# B&R Automation Studio project ComauRacer3demo (part 3)

### Main.st - not listed in the package file held
```iecst
PROGRAM _INIT
	cmd.MpFileManagerUI_0.MpLink := ADR(gFileManagerUI);
	cmd.MpFileManagerUI_0.Enable := TRUE;

	cmd.MpFileManagerUI_0.UISetup := cmd.MpFileManagerUISetupType;
	cmd.MpFileManagerUI_0.UIConnect := ADR(cmd.MpFileManagerUIConnectType);

	(* define of device names *)
	cmd.MpFileManagerUIConnectType.DeviceList.DeviceNames[0] := 'CNC_PrgDir';
	cmd.MpFileManagerUIConnectType.DeviceList.DeviceNames[1] := 'UserPart';
	cmd.MpFileManagerUIConnectType.DeviceList.DeviceNames[2] := 'AUDIT';
	cmd.MpFileManagerUIConnectType.DeviceList.DeviceNames[3] := 'RECIPE'; //currently not implemented

	cmd.MpFileManagerUIConnectType.File.NewName := '';

	cmd.MpFileManagerUI_0();
END_PROGRAM

PROGRAM _CYCLIC
	tabInfo.NumberOfElements := 0;
	FOR iFile := 0 TO 49 BY 1 DO
		(* create arrays with file properties *)
		brsmemcpy(ADR(tabInfo.Name[iFile]), ADR(cmd.MpFileManagerUIConnectType.File.List.Items[iFile].Name), SIZEOF(tabInfo.Name[iFile]));
		brsmemcpy(ADR(tabInfo.Size[iFile]), ADR(cmd.MpFileManagerUIConnectType.File.List.Items[iFile].Size), SIZEOF(tabInfo.Size[iFile]));
		brsmemcpy(ADR(tabInfo.Type[iFile]), ADR(cmd.MpFileManagerUIConnectType.File.List.Items[iFile].ItemType), SIZEOF(tabInfo.Type[iFile]));
		brsmemcpy(ADR(tabInfo.LastModified[iFile]), ADR(cmd.MpFileManagerUIConnectType.File.List.Items[iFile].LastModified), SIZEOF(tabInfo.LastModified[iFile]));

		IF tabInfo.SelectedRow = iFile THEN
			cmd.MpFileManagerUIConnectType.File.List.Items[iFile].IsSelected := TRUE;
		END_IF

		(* numbers of elements in the table *)
		IF tabInfo.Type[iFile] <> mpFILE_ITEM_TYPE_NONE THEN
			tabInfo.NumberOfElements := tabInfo.NumberOfElements + 1;
		END_IF
	END_FOR

	(* dynamic change of the array size *)
	brsitoa(tabInfo.NumberOfElements, ADR(aux.NumberOfElementsStr));
	aux.TableConfigurationStr := '{"specRows": [ {"from":0, "to":';
	aux.One := ', "visible":true}, {"from":';
	aux.Two := ', "to":49, "visible":false}]}';
	brsstrcat(ADR(aux.TableConfigurationStr), ADR(aux.NumberOfElementsStr));
	brsstrcat(ADR(aux.TableConfigurationStr), ADR(aux.One));
	brsstrcat(ADR(aux.TableConfigurationStr), ADR(aux.NumberOfElementsStr));
	brsstrcat(ADR(aux.TableConfigurationStr), ADR(aux.Two));

	aux.NumberOfElementsMinus := tabInfo.NumberOfElements - 1;

	IF tabInfo.NumberOfElements >= 1 THEN
		aux.NewNamePlus := 0;
		aux.newNewName := '';
		aux.prevNewName := cmd.MpFileManagerUIConnectType.File.NewName;
		aux.newNewName := aux.prevNewName;
		FOR iFile := 0 TO aux.NumberOfElementsMinus BY 1 DO
			(* dynamic change of the existing name *)
			IF tabInfo.Name[iFile] = aux.newNewName THEN
				aux.newNewName := aux.prevNewName;
				aux.NewNamePlus := aux.NewNamePlus + 1;
				brsitoa(aux.NewNamePlus, ADR(aux.NewNamePlusStr));
				aux.NewNameTextOne := '(';
				aux.NewNameTextTwo := ')';
				brsstrcat(ADR(aux.newNewName), ADR(aux.NewNameTextOne));
				brsstrcat(ADR(aux.newNewName), ADR(aux.NewNamePlusStr));
				brsstrcat(ADR(aux.newNewName), ADR(aux.NewNameTextTwo));
				//iFile := 0;
			ELSE
				cmd.MpFileManagerUIConnectType.File.NewName := aux.newNewName;
			END_IF
		END_FOR
	END_IF

	(* search engine *)
	cmd.MpFileManagerUIConnectType.File.Filter := '*';
	IF aux.SearchNewName <> '' THEN
		brsstrcat(ADR(cmd.MpFileManagerUIConnectType.File.Filter), ADR(aux.SearchNewName));
		brsstrcat(ADR(cmd.MpFileManagerUIConnectType.File.Filter), ADR(aux.textStar));
		cmd.MpFileManagerUIConnectType.File.Refresh := TRUE;
	ELSE
		cmd.MpFileManagerUIConnectType.File.Filter := '*';
	END_IF

	//change sorting method
	CASE aux.btnSort OF
		0:
			cmd.MpFileManagerUIConnectType.File.SortOrder := mpFILE_SORT_BY_NAME_ASC;
			aux.btnSortStr := '$$IAT/Browser/SortByNameAsc';
		1:
			cmd.MpFileManagerUIConnectType.File.SortOrder := mpFILE_SORT_BY_NAME_DESC;
			aux.btnSortStr := '$$IAT/Browser/SortByNameDesc';
		2:
			cmd.MpFileManagerUIConnectType.File.SortOrder := mpFILE_SORT_BY_SIZE_ASC;
			aux.btnSortStr := '$$IAT/Browser/SortBySizeAsc';
		3:
			cmd.MpFileManagerUIConnectType.File.SortOrder := mpFILE_SORT_BY_SIZE_DES;
			aux.btnSortStr := '$$IAT/Browser/SortBySizeDesc';
		4:
			cmd.MpFileManagerUIConnectType.File.SortOrder := mpFILE_SORT_BY_MOD_TIME_ASC;
			aux.btnSortStr := '$$IAT/Browser/SortByLastModAsc';
		5:
			cmd.MpFileManagerUIConnectType.File.SortOrder := mpFILE_SORT_BY_MOD_TIME_DESC;
			aux.btnSortStr := '$$IAT/Browser/SortByLastModDesc';
		6:
			aux.btnSort := 0;
	END_CASE

	//variables used to load files
	aux.fileName := tabInfo.Name[tabInfo.SelectedRow];
	aux.NewNameTextOne := '/';
	aux.fullFilePath := '';
	aux.fullFilePathWithFileDevice := '/FileDevice:';
	IF brsstrcmp(ADR(aux.fullFilePath), ADR(cmd.MpFileManagerUIConnectType.File.PathInfo.CurrentDir)) = 0 THEN //theoritically it works without it, but adds two '//' when not in a subfolder
		brsstrcat(ADR(aux.fullFilePath), ADR(cmd.MpFileManagerUIConnectType.DeviceList.DeviceNames[cmd.MpFileManagerUIConnectType.DeviceList.SelectedIndex])); //device name
		brsstrcat(ADR(aux.fullFilePath), ADR(aux.NewNameTextOne)); // '/'
		brsstrcat(ADR(aux.fullFilePath), ADR(aux.fileName)); // file name, this gives full file path in subsystem.
	ELSE
		brsstrcat(ADR(aux.fullFilePath), ADR(cmd.MpFileManagerUIConnectType.DeviceList.DeviceNames[cmd.MpFileManagerUIConnectType.DeviceList.SelectedIndex])); //device name
		brsstrcat(ADR(aux.fullFilePath), ADR(aux.NewNameTextOne)); // '/'
		brsstrcat(ADR(aux.fullFilePath), ADR(cmd.MpFileManagerUIConnectType.File.PathInfo.CurrentDir)); //this adds subfolder compatibility
		brsstrcat(ADR(aux.fullFilePath), ADR(aux.NewNameTextOne)); // '/'
		brsstrcat(ADR(aux.fullFilePath), ADR(aux.fileName)); // file name, this gives full file path in subsystem.
	END_IF

	brsstrcat(ADR(aux.fullFilePathWithFileDevice), ADR(aux.fullFilePath)); //this gives variable with /FileDevice: prefix, used for PDFs and images.

	aux.fileExtension3Chars; //PDF detection
	brsmemcpy(ADR(aux.fileExtension3Chars), ADR(aux.fileName)+brsstrlen(ADR(aux.fileName))-4, 4);
	IF (brsstrcmp(ADR(aux.fileExtension3Chars), ADR(aux.fileExtensionPDF)) = 0) OR (brsstrcmp(ADR(aux.fileExtension3Chars), ADR(aux.fileExtensionpdf)) = 0) THEN
		aux.IsPDF := TRUE;

	ELSE
		aux.IsPDF := FALSE;
	END_IF

	cmd.MpFileManagerUI_0();
END_PROGRAM

PROGRAM _EXIT
	(* Insert code here *)
	cmd.MpFileManagerUI_0.Enable := FALSE;
	cmd.MpFileManagerUI_0();
END_PROGRAM
```

### Program Logical/Audit

#### Variables.var
```iecst
VAR
	MpAuditTrail_0 : MpAuditTrail;
	TriggerEvent : BOOL;
	TypeVar : WSTRING[100];
	MessageVar : WSTRING[100];
	CommentVar : WSTRING[100];
	CustomEventStatus : DINT;
END_VAR
```

#### Main.st
```iecst
PROGRAM _INIT
	MpAuditTrail_0.Enable := TRUE;
	MpAuditTrail_0.MpLink := ADR(gAuditTrail);
	MpAuditTrail_0.DeviceName := ADR('CF');
	MpAuditTrail_0.Language := ADR('en|metric');
END_PROGRAM

PROGRAM _CYCLIC

	MpAuditTrail_0();

	IF(TriggerEvent)THEN
		CustomEventStatus := MpAuditCustomEvent(MpLink := gAuditTrail, Type := TypeVar, Message := MessageVar, Comment := CommentVar);
		TriggerEvent := FALSE;
	END_IF

END_PROGRAM

PROGRAM _EXIT
	MpAuditTrail_0.Enable := FALSE;
	MpAuditTrail_0();
END_PROGRAM
```

### Program Logical/Audit_notworking

#### Main.st
```iecst
PROGRAM _INIT
	MpAuditTrail_0.Enable := TRUE;
	MpAuditTrail_0.MpLink := ADR(gAuditTrail);
	MpAuditTrail_0.DeviceName := ADR('CF');
	MpAuditTrail_0.Language := ADR('end|metric');
END_PROGRAM

PROGRAM _CYCLIC

	MpAuditTrail_0();

	IF(TriggerEvent)THEN
		CustomEventStatus := MpAuditCustomEvent(MpLink := gAuditTrail, Type := TypeVar, Message := MessageVar, Comment := CommentVar);
		TriggerEvent := FALSE;
	END_IF

END_PROGRAM

PROGRAM _EXIT
	MpAuditTrail_0.Enable := FALSE;
	MpAuditTrail_0();
END_PROGRAM
```

### Program Logical/Program

#### Variables.var
```iecst
VAR
	RoboArm6AxisPara : MpRoboArm6AxisParType;
	RoboArm6Axis : MpRoboArm6Axis;
	ManualMode : R3ManualModeType;
	j : INT;
END_VAR
```

#### Main.st
```iecst
PROGRAM _INIT

	RoboArm6Axis.Enable := TRUE;

	RoboArm6Axis.Override  := 100.0;
	RoboArm6AxisPara.ProgramName := 'Robotic.st';    //File stored on FileDevice
	RoboArm6Axis.MpLink     := ADR(gAxesGroupRacer3);
	RoboArm6Axis.Parameters := ADR(RoboArm6AxisPara);
	RoboArm6AxisPara.Acceleration := 1000.0;
	RoboArm6AxisPara.Deceleration := 1000.0;
	RoboArm6AxisPara.Velocity := 100.0;
	//RoboArm6AxisPara.Distance[0] := 50.0;
	ManualMode.PathLimits.Acceleration := 100.0;
	ManualMode.CoordinateSystem := 9;
	ManualMode.PathLimits.Deceleration := 100.0;
	ManualMode.PathLimits.Velocity := 10.0;
	ManualMode.PathLimits.Jerk := 0.0;
	ManualMode.Direction := POSITIVE;

END_PROGRAM

PROGRAM _CYCLIC

	RoboArm6AxisPara.Jog.CoordSystem := ManualMode.CoordinateSystem;
	RoboArm6AxisPara.Jog.PathLimits := ManualMode.PathLimits;

	IF RoboArm6Axis.Info.ReadyToPowerOn THEN

		RoboArm6Axis.Power := TRUE;

		IF RoboArm6Axis.PowerOn THEN

			IF ManualMode.Direction = POSITIVE THEN // set actual axis velocity based on which direction it's set to be moved
				ManualMode.JogVelocityActual := ManualMode.JogVelocity;
			ELSIF ManualMode.Direction = NEGATIVE THEN
				ManualMode.JogVelocityActual := -1 * ManualMode.JogVelocity;
			END_IF

			IF ManualMode.AxisButton.Q1 THEN // if a button is pressed, write corresponding velocity to the jog velocity array
				RoboArm6AxisPara.Jog.Velocity[0] := ManualMode.JogVelocityActual;
				RoboArm6Axis.Jog := TRUE;
			ELSIF ManualMode.AxisButton.Q2 THEN
				RoboArm6AxisPara.Jog.Velocity[1] := ManualMode.JogVelocityActual;
				RoboArm6Axis.Jog := TRUE;
			ELSIF ManualMode.AxisButton.Q3 THEN
				RoboArm6AxisPara.Jog.Velocity[2] := ManualMode.JogVelocityActual;
				RoboArm6Axis.Jog := TRUE;
			ELSIF ManualMode.AxisButton.Q4 THEN
				RoboArm6AxisPara.Jog.Velocity[3] := ManualMode.JogVelocityActual;
				RoboArm6Axis.Jog := TRUE;
			ELSIF ManualMode.AxisButton.Q5 THEN
				RoboArm6AxisPara.Jog.Velocity[4] := ManualMode.JogVelocityActual;
				RoboArm6Axis.Jog := TRUE;
			ELSIF ManualMode.AxisButton.Q6 THEN
				RoboArm6AxisPara.Jog.Velocity[5] := ManualMode.JogVelocityActual;
				RoboArm6Axis.Jog := TRUE;
			ELSE //if no buttons are pressed reset jog velocity array
				RoboArm6Axis.Jog := FALSE;
				FOR j := 0 TO 5 BY 1 DO //set every jog velocity to 0
					RoboArm6AxisPara.Jog.Velocity[j] := 0.0;
				END_FOR;
			END_IF

		END_IF
	END_IF

	IF RoboArm6Axis.UpdateDone THEN
		RoboArm6Axis.Update := FALSE;
	END_IF

	IF NOT RoboArm6Axis.Error THEN
		RoboArm6Axis.ErrorReset := FALSE;
	END_IF

	RoboArm6Axis();
END_PROGRAM

PROGRAM _EXIT
	(* Insert code here *)

END_PROGRAM
```

### Program Logical/Program1

#### Variables.var
```iecst
VAR
	test : BOOL;
END_VAR
```

#### Main.st
```iecst
PROGRAM _INIT
	(* Insert code here *)
	 test := FALSE;
END_PROGRAM

PROGRAM _CYCLIC
	(* Insert code here *)
	 test := TRUE;
END_PROGRAM

PROGRAM _EXIT
	(* Insert code here *)

END_PROGRAM
```

### Program Logical/Recipe

#### Variables.var
```iecst
VAR
	R3AutomaticModePara_Recipe : R3AutomaticModePara;
	CalibrationParaType_Recipe : CalibrationParaType;
	MpRecipeXml_0 : MpRecipeXml;
END_VAR
```

#### Main.st
```iecst
PROGRAM _INIT
	MpRecipeXml_0(MpLink := ADR(gRecipeXmlLink), Enable := FALSE, ErrorReset := TRUE, DeviceName := ADR('RECIPE') , FileName := ADR('Recipe_0'));
END_PROGRAM

PROGRAM _CYCLIC
		MpRecipeXml_0(Enable :=TRUE);
END_PROGRAM

PROGRAM _EXIT
	(* Insert code here *)

END_PROGRAM
```

Listed in the project but not available here: Logical/Libraries/RacerLib/ManualCtrl/Types.typ, Logical/Libraries/RacerLib/ManualCtrl/Constants.var
